TYPE ST_MachineSetting :
STRUCT
//	astWorkpiecePlaceStates					: ARRAY[0..GVL.nMaxWorkpiecePlaceStatus] OF TcaWorkpiecePlaceStatus;
//	astWorkpieceType						: ARRAY[0..GVL.nMaxWorkpieceTyp] OF ST_WorkpieceType;
END_STRUCT
END_TYPE

(* stored: Version 1.1.0.1
   DUT ST_MachineSetting: Id {8f809027-6a1f-4e9a-b552-63efee118c54} *)
